(* IEC 61131-3 sources: Caravan/Archiv/12-04-19/Stations/MachineControl/MachineControl/Class/HmiSetupList35, 1 file *)

(* ---- HmiSetupList35.st ---- *)
(*!
<Class
	Name               = "HmiSetupList35"
	Revision           = "0.2"
	RealtimeTask       = "false"
	CyclicTask         = "false"
	BackgroundTask     = "false"
	Sigmatek           = "true"
	OSInterface        = "false"
	HighPriority       = "false"
	Automatic          = "false"
	UpdateMode         = "Prescan"
	SharedCommandTable = "true"
	Objectsize         = "(284,120)">
	<Channels>
		<Server Name="ClassSvr" Visualized="false" Initialize="false" WriteProtected="true" Retentive="false"/>
	</Channels>
	<RevDoku>
		<Owner Company="sigmatek" Author="kolott"/>
		<Dokumentation Revision="0.2" Date="2018-05-24" Author="kolott" Company="sigmatek" Description="sa41119, devsw-502: modification of method Create() to send Setup Standardfonts as well to HMI"/>
		<Dokumentation Revision="0.1" Date="2017-11-27" Author="kolott" Company="sigmatek" Description="projectversion will be sent to hmi as well"/>
	</RevDoku>
</Class>
*)
HmiSetupList35 : CLASS
  //Servers:
	ClassSvr 	: SvrChCmd_DINT;
  //Clients:
  //Variables:
		xData : ARRAY [0..2000] OF USINT;

  //Functions:

	FUNCTION GLOBAL Start;

	FUNCTION GLOBAL End
		VAR_OUTPUT
			retcode 	: ^void;
		END_VAR;

	FUNCTION GLOBAL Create
		VAR_INPUT
			color_button 	: UINT;
			color_button_text 	: UINT;
			color_title_text 	: UINT;
			color_limit_text 	: UINT;
			color_window 	: UINT;
			frame_button 	: USINT;
			frame_window 	: USINT;
			user_prj_revision 	: UINT;
			font_std 	: USINT;
			font_std_small 	: USINT;
		END_VAR;
  //Tables:
	FUNCTION @STD
		VAR_OUTPUT
			ret_code	: CONFSTATES;
		END_VAR;
	FUNCTION GLOBAL TAB @CT_;
END_CLASS;

#includeC "..\LseEasy\Create.h"

FUNCTION GLOBAL HmiSetupList35::Start
  var
    pbox : ^_BOX_SETUPLIST;
  end_var

  pbox$^usint := #xData[0];
  pbox^.boxhdr.crc32 := 0;
  pbox^.boxhdr.size  := 0;

END_FUNCTION

FUNCTION GLOBAL HmiSetupList35::End
	VAR_OUTPUT
		retcode 	: ^void;
	END_VAR
  var
    pbox : ^_BOX_SETUPLIST;
  end_var

  pbox$^usint := #xData[0];
  ClassSvr    := 1;
  end_BIGBOX_HEADER(#pbox^.boxhdr, sizeof(_BOX_SETUPLIST));

  retcode := pbox;

END_FUNCTION

FUNCTION GLOBAL HmiSetupList35::Create
	VAR_INPUT
		color_button 	: UINT;
		color_button_text 	: UINT;
		color_title_text 	: UINT;
		color_limit_text 	: UINT;
		color_window 	: UINT;
		frame_button 	: USINT;
		frame_window 	: USINT;
		user_prj_revision 	: UINT;
		font_std 	: usint;
		font_std_small 	: usint;
	END_VAR
  var
    pbox : ^_BOX_SETUPLIST;
  end_var

  pbox$^usint := #xData[0];

  _memset(#xData[0], 0, sizeof(_BOX_SETUPLIST));

  pbox^.color_button      := color_button;      // color of button
  pbox^.color_button_text := color_button_text; // color of buttontext
  pbox^.color_title_text  := color_title_text;  // color of titletext
  pbox^.color_limit_text  := color_limit_text;  // color of limittext
  pbox^.color_window      := color_window;      // backgroundcolor
  pbox^.button_frametype  := frame_button;      // frametype button
  pbox^.window_frametype  := frame_window;      // frametype window
  pbox^.user_prj_revision := user_prj_revision; // user-project-revision
  pbox^.font_standard     := font_std;
  pbox^.font_standard_small := font_std_small;

END_FUNCTION
